// TIA Portal V20 export
// export: Created 2025-12-01T14:57:08.3295832Z, ExportSetting None, DisplayName Totally Integrated Automation Portal, DisplayVersion V20 Update 3, DisplayName TIA Portal Openness, DisplayVersion V20 Update 3, DisplayName TIA Portal Version Control Interface, DisplayVersion V20 Update 3, DisplayName STEP 7 Professional, DisplayVersion V20 Update 3, DisplayName STEP 7 Safety, DisplayVersion V20 Update 2, DisplayName WinCC Basic/Comfort/Advanced, DisplayVersion V20 Update 3, DisplayName WinCC Professional, DisplayVersion V20 Update 3, DisplayName WinCC Unified, DisplayVersion V20 Update 3
FUNCTION "FC825_CalcularOrdenUT_MesaPaso" : Void   // FC825, STL
{ S7_Optimized_Access := 'FALSE' }
// stored: AutoNumber false
   VAR_INPUT
      NumeroUT : UInt;
   END_VAR
   VAR_OUTPUT
      Orden : Word;   // Orden a realizar en la MESA
      Auxiliar_01 : UInt;   // Auxiliar 01 de la Orden a realizar en la MESA
      MesaSalidaMulti : UInt;   // Auxiliar 02 de la Orden a realizar en la MESA
      Auxiliar_03 : UInt;   // Auxiliar 03 de la Orden a realizar en la MESA
      Auxiliar_04 : UInt;   // Auxiliar 04 de la Orden a realizar en la MESA
   END_VAR
   VAR_TEMP
      P_Temporal : DWord;
      NumeroMesa : UInt;
      SiguienteUT : UInt;
      MesaEspera : UInt;
      OrdenTMP : Word;
      SinUT_EnMesa : Bool;
      RutaOK_EnMesa : Bool;
   END_VAR
BEGIN

NETWORK
TITLE = Inicializar
/////////////////////////////////////////////////////////////////////////
// Inicializaciones de las variables de los DB's

      L     0;
      T     #Orden;
      T     #OrdenTMP;
      T     #MesaSalidaMulti;
      T     #Auxiliar_01;
      T     #Auxiliar_03;
      T     #Auxiliar_04;


/////////////////////////////////////////////////////////////////////////
// Mesa Actual dentro del PLC
      L     "DB812_UTs_Control".UT[#NumeroUT].MesaActual;
      L     "CTE_OffsetMesa";
      -I;
      T     #NumeroMesa;



NETWORK
TITLE = Calcular Orden - FASE 01 >>> Tiene Libre el Camnino
/////////////////////////////////////////////////////////////////////////
// --- Es una Mesa de Paso (Un solo camino posible)
/////////////////////////////////////////////////////////////////////////
// Condiciones:
//
// - Para enviar orden hay que ver si tiene que ESPERAR a que este LIBRE la
//   mesa SIGUIENTE (Mesa_Sxx) dependiendo de la salida definida
//
// - Si tiene que esperar, no hacer nada
// - Si no tiene que esperar, enviar orden y darla por tratada
//
/////////////////////////////////////////////////////////////////////////


/////////////////////////////////////////////////////////////////////////
/////////////////////////////////////////////////////////////////////////
/////////////////////////////////////////////////////////////////////////
// --- FASE 01, Mirar si la mesa esta definido como ESPERA

      SET;
      AN    "DB850_DefinicionMesas".Mesa[#NumeroMesa].ConfigMesa.Espera_S01;
      AN    "DB850_DefinicionMesas".Mesa[#NumeroMesa].ConfigMesa.Espera_S02;
      AN    "DB850_DefinicionMesas".Mesa[#NumeroMesa].ConfigMesa.Espera_S03;
      AN    "DB850_DefinicionMesas".Mesa[#NumeroMesa].ConfigMesa.Espera_S04;
      JC    FinalControlEnMesaEspera;


/////////////////////////////////////////////////////////////////////////
// --- Ver si la que esta definida es la Mesa S01
      SET;
      AN    "DB850_DefinicionMesas".Mesa[#NumeroMesa].ConfigMesa.Espera_S01;
      JC    FinalEnMesaEspera_S01;

      L     "DB850_DefinicionMesas".Mesa[#NumeroMesa].Mesa_S01;
      L     "CTE_OffsetMesa";
      -I;  // --- Calculo de la Mesa en Espera 28/03/2022
      T     #MesaEspera;

      CALL  "FC870_MesaSinUT"
      ( Mesa  := #MesaEspera,
        SinUT := #SinUT_EnMesa
      );

      SET;  // Mesa esta sin UT ?
      A     "DB850_DefinicionMesas".Mesa[#NumeroMesa].ConfigMesa.Espera_S01;
      A     #SinUT_EnMesa;
      JC    FinalControlEnMesaEspera;
// Mesa esta con UT ?
      JU    FinalCalcularOrden;

FinalEnMesaEspera_S01:NOP   0;


/////////////////////////////////////////////////////////////////////////
// --- Ver si la que esta definida es la Mesa S02
      SET;
      AN    "DB850_DefinicionMesas".Mesa[#NumeroMesa].ConfigMesa.Espera_S02;
      JC    FinalEnMesaEspera_S02;

      L     "DB850_DefinicionMesas".Mesa[#NumeroMesa].Mesa_S02;
      L     "CTE_OffsetMesa";
      -I;  // --- Calculo de la Mesa en Espera 28/03/2022
      T     #MesaEspera;

      CALL  "FC870_MesaSinUT"
      ( Mesa  := #MesaEspera,
        SinUT := #SinUT_EnMesa
      );

      SET;  // Mesa esta sin UT ?
      A     "DB850_DefinicionMesas".Mesa[#NumeroMesa].ConfigMesa.Espera_S02;
      A     #SinUT_EnMesa;
      JC    FinalControlEnMesaEspera;
// Mesa esta con UT ?
      JU    FinalCalcularOrden;

FinalEnMesaEspera_S02:NOP   0;


/////////////////////////////////////////////////////////////////////////
// --- Ver si la que esta definida es la Mesa S03
      SET;
      AN    "DB850_DefinicionMesas".Mesa[#NumeroMesa].ConfigMesa.Espera_S03;
      JC    FinalEnMesaEspera_S03;

      L     "DB850_DefinicionMesas".Mesa[#NumeroMesa].Mesa_S03;
      L     "CTE_OffsetMesa";
      -I;  // --- Calculo de la Mesa en Espera 28/03/2022
      T     #MesaEspera;

      CALL  "FC870_MesaSinUT"
      ( Mesa  := #MesaEspera,
        SinUT := #SinUT_EnMesa
      );

      SET;  // Mesa esta sin UT ?
      A     "DB850_DefinicionMesas".Mesa[#NumeroMesa].ConfigMesa.Espera_S03;
      A     #SinUT_EnMesa;
      JC    FinalControlEnMesaEspera;
// Mesa esta con UT ?
      JU    FinalCalcularOrden;

FinalEnMesaEspera_S03:NOP   0;


/////////////////////////////////////////////////////////////////////////
// --- Ver si la que esta definida es la Mesa S04
      SET;
      AN    "DB850_DefinicionMesas".Mesa[#NumeroMesa].ConfigMesa.Espera_S04;
      JC    FinalEnMesaEspera_S04;

      L     "DB850_DefinicionMesas".Mesa[#NumeroMesa].Mesa_S04;
      L     "CTE_OffsetMesa";
      -I;  // --- Calculo de la Mesa en Espera 28/03/2022
      T     #MesaEspera;

      CALL  "FC870_MesaSinUT"
      ( Mesa  := #MesaEspera,
        SinUT := #SinUT_EnMesa
      );

      SET;  // Mesa esta sin UT ?
      A     "DB850_DefinicionMesas".Mesa[#NumeroMesa].ConfigMesa.Espera_S04;
      A     #SinUT_EnMesa;
      JC    FinalControlEnMesaEspera;
// Mesa esta con UT ?
      JU    FinalCalcularOrden;

FinalEnMesaEspera_S04:NOP   0;


/////////////////////////////////////////////////////////////////////////
// La UT Tiene Camino Libre - Final de FASE 01
FinalControlEnMesaEspera:NOP   0;




NETWORK
TITLE = Calcular Orden - FASE 02 >>> Tiene Ruta Para Continuar
/////////////////////////////////////////////////////////////////////////
/////////////////////////////////////////////////////////////////////////
/////////////////////////////////////////////////////////////////////////
// --- FASE 02, Mirar las rutas de las UT's de la Mesa
      SET;
      A     "DB850_DefinicionMesas".Mesa[#NumeroMesa].ConfigMesa.RutaSalidaTodas;
      O     "DB850_DefinicionMesas".Mesa[#NumeroMesa].ConfigMesa.MultiplesCargasDeSalida;
      O     "DB850_DefinicionMesas".Mesa[#NumeroMesa].ConfigMesa.GrupoDeSalida;
      JCN   FinalControlRutaEnMesa;

      CALL  "FC872_VerificarRutaEnMesa"
      ( Mesa      := #NumeroMesa,
        TestGrupo := "DB850_DefinicionMesas".Mesa[#NumeroMesa].ConfigMesa.GrupoDeSalida,
        RutaOK    := #RutaOK_EnMesa
      );

      SET;  // No tienen todas Ruta ?
      AN    #RutaOK_EnMesa;
      JC    FinalCalcularOrden;

/////////////////////////////////////////////////////////////////////////
// Tiene Ruta para Continuar - Final de FASE 02
FinalControlRutaEnMesa:NOP   0;



NETWORK
TITLE = Calcular Orden - FASE 03 >>> Final, Calcular la Salida de la Mesa
/////////////////////////////////////////////////////////////////////////
/////////////////////////////////////////////////////////////////////////
/////////////////////////////////////////////////////////////////////////
// --- FASE 03, Se envia orden
// --- Mirando que mesa esta definida (Solo puede haber una)
// --- Primero, doy por tratada la causa
// --- Segundo, mirar que salida debe activarse
// ---          sino hay ninguna mesa definida no se envia la orden


/////////////////////////////////////////////////////////////////////////
// --- Doy por tratada la Mesa la Primera de la Mesa
      L     0;  // Dar por tratada
      T     "DB812_UTs_Control".UT[#NumeroUT].EstadoRecepcionUT;
      T     "DB812_UTs_Control".UT[#NumeroUT].EstadoEventoRecibido;


/////////////////////////////////////////////////////////////////////////
// --- Si hay que darla por tratadas todas las de la Mesa

      SET;  // Hay que Recorrer el Resto de UTs de la Mesa
      AN    "DB850_DefinicionMesas".Mesa[#NumeroMesa].ConfigMesa.MultiplesCargasDeSalida;
      AN    "DB850_DefinicionMesas".Mesa[#NumeroMesa].ConfigMesa.GrupoDeSalida;
      JC    FinalBucleUTs_EnMesa;

      L     "DB812_UTs_Control".UT[#NumeroUT].UT_SiguienteMesa;
      T     #SiguienteUT;

InicioBucleUTs_EnMesa:NOP   0;
      L     #SiguienteUT;
      L     0;
      ==I;  // Hay mas UT's
      JC    FinalBucleUTs_EnMesa;

// Testear Grupo ?
      SET;
      AN    "DB850_DefinicionMesas".Mesa[#NumeroMesa].ConfigMesa.GrupoDeSalida;
      JC    ContinuarBucleUTs_EnMesa;

// Dar por tratado solo lo del mismo Grupo
// Grupo Primera UT == Grupo de la Siguiente
      L     "DB812_UTs_Control".UT[#NumeroUT].Grupo;
      L     "DB812_UTs_Control".UT[#SiguienteUT].Grupo;
      <>I;
      JC    FinalBucleUTs_EnMesa;

// Dar por tratada la Siguinete UT
ContinuarBucleUTs_EnMesa:NOP   0;
      L     0;  // Dar por tratada
      T     "DB812_UTs_Control".UT[#SiguienteUT].EstadoRecepcionUT;
      T     "DB812_UTs_Control".UT[#SiguienteUT].EstadoEventoRecibido;

      L     "DB812_UTs_Control".UT[#SiguienteUT].UT_SiguienteMesa;
      T     #SiguienteUT;
      JU    InicioBucleUTs_EnMesa;


/////////////////////////////////////////////////////////////////////////
// Final del Bucle
FinalBucleUTs_EnMesa:NOP   0;




/////////////////////////////////////////////////////////////////////////
// --- Mirar que salida esta activa, solo tiene una salida posible (MesaPaso)
//     La Primera definida
// --- Sino se define ninguna mesa, no se enviara Orden

      L     "DB850_DefinicionMesas".Mesa[#NumeroMesa].Mesa_S01;
      L     0;
      <>I;  // Esta definida la Mesa S01
      JC    OrdenSalida_S01;

      L     "DB850_DefinicionMesas".Mesa[#NumeroMesa].Mesa_S02;
      L     0;
      <>I;  // Esta definida la Mesa S02
      JC    OrdenSalida_S02;

      L     "DB850_DefinicionMesas".Mesa[#NumeroMesa].Mesa_S03;
      L     0;
      <>I;  // Esta definida la Mesa S03
      JC    OrdenSalida_S03;

      L     "DB850_DefinicionMesas".Mesa[#NumeroMesa].Mesa_S04;
      L     0;
      <>I;  // Esta definida la Mesa S04
      JC    OrdenSalida_S04;

/////////////////////////////////////////////////////////////////////////
// NUEVA OPERATIVA 2016 05 25 (Alonso)
// --- Sino se define ninguna mesa, no se enviara Orden
      JU    FinalCalcularOrden;



NETWORK
TITLE = Generar Orden de Salida
/////////////////////////////////////////////////////////////////////////
/////////////////////////////////////////////////////////////////////////
// --- Ordenes a enviar dependiendo por donde sale
// --- Salida por S01
OrdenSalida_S01:NOP   0;
      L     P##OrdenTMP;
      L     P#0.1;
      +D;
      T     #P_Temporal;

      SET;  // Orden -> Activar Bit 1
      S     L [#P_Temporal];
      JU    FinalOrdenSalida;


/////////////////////////////////////////////////////////////////////////
/////////////////////////////////////////////////////////////////////////
// --- Ordenes a enviar dependiendo por donde sale
// --- Salida por S02
OrdenSalida_S02:NOP   0;
      L     P##OrdenTMP;
      L     P#0.2;
      +D;
      T     #P_Temporal;

      SET;  // Orden -> Activar Bit 2
      S     L [#P_Temporal];
      JU    FinalOrdenSalida;


/////////////////////////////////////////////////////////////////////////
/////////////////////////////////////////////////////////////////////////
// --- Ordenes a enviar dependiendo por donde sale
// --- Salida por S03
OrdenSalida_S03:NOP   0;
      L     P##OrdenTMP;
      L     P#0.3;
      +D;
      T     #P_Temporal;

      SET;  // Orden -> Activar Bit 3
      S     L [#P_Temporal];
      JU    FinalOrdenSalida;


/////////////////////////////////////////////////////////////////////////
/////////////////////////////////////////////////////////////////////////
// --- Ordenes a enviar dependiendo por donde sale
// --- Salida por S04
OrdenSalida_S04:NOP   0;
      L     P##OrdenTMP;
      L     P#0.4;
      +D;
      T     #P_Temporal;

      SET;  // Orden -> Activar Bit 4
      S     L [#P_Temporal];
      JU    FinalOrdenSalida;



/////////////////////////////////////////////////////////////////////////
/////////////////////////////////////////////////////////////////////////
// --- Ordenes a enviar dependiendo por donde sale
// --- Salida por Defecto
OrdenSalida_Defecto:NOP   0;
      L     P##OrdenTMP;
      L     P#0.5;
      +D;
      T     #P_Temporal;

      SET;  // Orden -> Activar Bit 5
      S     L [#P_Temporal];
      JU    FinalOrdenSalida;


/////////////////////////////////////////////////////////////////////////
/////////////////////////////////////////////////////////////////////////
// No Existen mas posibilidades
FinalOrdenSalida:NOP   0;



NETWORK
TITLE = Final de Calcular Orden
/////////a////////////////////////////////////////////////////////////////
// Finalizar la Funcion
FinalCalcularOrden:NOP   0;

      L     #OrdenTMP;
      T     #Orden;


END_FUNCTION
